Yaskawa INFORM job: 34.JBI

/JOB
//NAME 34
//POS
///NPOS 208,208,208,10,0,0
///TOOL 0
///POSTYPE PULSE
///PULSE
C00000=-36470,-76528,-106815,19279,71473,77234
C00001=-134470,-76528,-106815,19279,71473,77234
C00002=-159578,-94739,-111578,14965,102577,71346
C00003=-157881,-88069,-71686,3941,80760,68512
C00004=-158562,-88051,-67559,4028,78269,68198
C00005=-158841,-87937,-65852,4065,77294,68070
C00006=-158823,-87020,-63758,4076,76477,68050
C00007=-158841,-87937,-65852,4065,77294,68070
C00008=-158257,-85912,-63562,4020,76897,68259
C00009=-159408,-88670,-64664,4131,76218,67839
C00010=-158257,-85912,-63562,4020,76897,68259
C00011=-157986,-86044,-65280,3983,77870,68384
C00012=-157322,-86111,-69434,3896,80354,68691
C00013=-157948,-93050,-93119,3918,91369,68820
C00014=-158631,-94954,-89856,3971,88424,68498
C00015=-158911,-95544,-88477,3995,87288,68367
C00016=-158893,-95136,-86651,3995,86375,68344
C00017=-158911,-95544,-88477,3995,87288,68367
C00018=-158162,-93185,-86154,3931,87034,68613
C00019=-159307,-96640,-87495,4031,86143,68197
C00020=-158162,-93185,-86154,3931,87034,68613
C00021=-157891,-92621,-87539,3907,88161,68739
C00022=-157230,-90799,-90820,3855,91078,69051
C00023=-157971,-89638,-106553,4024,101368,69130
C00024=-158653,-94046,-104272,4030,97741,68787
C00025=-158932,-95549,-103251,4038,96357,68649
C00026=-158915,-95836,-101701,4026,95258,68619
C00027=-158932,-95549,-103251,4038,96357,68649
C00028=-158118,-93796,-101169,3964,95939,68906
C00029=-159263,-97999,-102797,4052,94839,68490
C00030=-158118,-93796,-101169,3964,95939,68906
C00031=-157847,-92365,-102209,3955,97297,69039
C00032=-157186,-88172,-104546,3946,100851,69371
C00033=-156260,-82084,-105550,20461,72444,69801
C00034=-137260,-84248,-120477,10166,77039,76482
C00035=11401,-148032,-125425,11667,16324,75771
C00036=126225,-114648,-117375,36487,17100,65054
C00037=168603,-127327,-105850,12339,78437,77405
C00038=188556,-88570,-70376,9474,73843,-79671
C00039=189658,-87934,-65982,9402,71368,-79472
C00040=190106,-87582,-64173,9375,70395,-79388
C00041=190093,-86631,-62058,9423,69594,-79456
C00042=190106,-87582,-64173,9375,70395,-79388
C00043=189092,-85833,-61994,9573,70077,-79779
C00044=190880,-87833,-62791,9297,69339,-79192
C00045=189092,-85833,-61994,9573,70077,-79779
C00046=188652,-86197,-63814,9595,71050,-79858
C00047=187573,-86869,-68234,9657,73522,-80046
C00048=174405,-91869,-88866,8360,85065,-80378
C00049=162023,-93599,-92534,7262,87848,-81242
C00050=162738,-95362,-89212,7186,84857,-81172
C00051=163031,-95900,-87810,7159,83700,-81138
C00052=163022,-95451,-85967,7171,82804,-81192
C00053=163031,-95900,-87810,7159,83700,-81138
C00054=162558,-93657,-85516,7221,83485,-81312
C00055=163728,-97065,-86834,7086,82448,-80971
C00056=162558,-93657,-85516,7221,83485,-81312
C00057=162272,-93147,-86925,7246,84631,-81343
C00058=161575,-91472,-90271,7318,87591,-81408
C00059=161833,-89597,-103823,7401,96799,-80781
C00060=162061,-91169,-106298,7358,97489,-80667
C00061=162777,-95345,-103917,7205,93844,-80645
C00062=163070,-96760,-102859,7152,92451,-80627
C00063=163061,-96969,-101279,7144,91380,-80691
C00064=163070,-96760,-102859,7152,92451,-80627
C00065=162549,-94558,-100616,7215,92250,-80812
C00066=163719,-98703,-102215,7058,91010,-80493
C00067=162549,-94558,-100616,7215,92250,-80812
C00068=162264,-93207,-101689,7266,93618,-80828
C00069=161567,-89224,-104115,7414,97191,-80847
C00070=161715,-86803,-103327,4886,98608,-77730
C00071=162141,-92472,-85533,-3463,86932,-68770
C00072=162126,-88781,-71814,-3762,80467,-68306
C00073=162843,-88708,-67661,-3852,77988,-67984
C00074=163137,-88572,-65944,-3890,77018,-67852
C00075=163128,-87638,-63844,-3901,76206,-67830
C00076=163137,-88572,-65944,-3890,77018,-67852
C00077=162593,-86370,-63634,-3847,76702,-68030
C00078=163767,-89113,-64727,-3960,76023,-67603
C00079=162593,-86370,-63634,-3847,76702,-68030
C00080=162306,-86518,-65359,-3809,77672,-68159
C00081=161607,-86627,-69532,-3720,80146,-68475
C00082=161949,-92223,-96357,-3744,93768,-68761
C00083=162073,-93836,-93212,-3726,91015,-68637
C00084=162789,-95666,-89915,-3783,88086,-68309
C00085=163083,-96227,-88523,-3809,86956,-68176
C00086=163074,-95793,-86687,-3810,86051,-68151
C00087=163083,-96227,-88523,-3809,86956,-68176
C00088=162687,-94151,-86288,-3775,86630,-68300
C00089=163864,-97585,-87612,-3878,85738,-67874
C00090=162687,-94151,-86288,-3775,86630,-68300
C00091=162400,-93622,-87691,-3749,87749,-68430
C00092=161699,-91892,-91016,-3692,90646,-68752
C00093=162002,-88104,-107646,-3859,102814,-69021
C00094=162113,-90810,-106745,-3822,100878,-68922
C00095=162829,-95111,-104412,-3836,97273,-68574
C00096=163122,-96572,-103371,-3847,95899,-68434
C00097=163114,-96817,-101805,-3837,94811,-68403
C00098=163122,-96572,-103371,-3847,95899,-68434
C00099=162678,-95201,-101447,-3805,95399,-68566
C00100=163858,-99394,-103055,-3897,94292,-68140
C00101=162678,-95201,-101447,-3805,95399,-68566
C00102=162391,-93819,-102511,-3793,96748,-68703
C00103=161689,-89747,-104911,-3775,100278,-69043
C00104=160138,-149166,-122708,-13309,73561,-68802
C00105=149595,-96211,-103761,-5489,101844,-74102
C00106=149594,-96505,-102316,-5465,100808,-74056
C00107=149006,-93113,-100988,-5479,101691,-74295
C00108=149599,-96300,-103483,-5484,101628,-74092
C00109=149598,-96527,-102324,-5465,100802,-74055
C00110=149603,-96557,-102335,-5465,100793,-74053
C00111=149607,-96579,-102343,-5465,100787,-74051
C00112=149608,-96287,-103789,-5489,101823,-74097
C00113=160720,-151449,-123129,-13814,72249,-68439
C00114=174899,-138237,-126795,1008,88740,-67536
C00115=163022,-96341,-102515,22398,105363,-76518
C00116=163017,-96713,-99258,22147,103326,-76913
C00117=163015,-96754,-97914,22060,102538,-77063
C00118=163022,-96736,-99152,22139,103253,-76925
C00119=162158,-93804,-96763,22109,103515,-77196
C00120=163010,-96735,-97907,22060,102545,-77064
C00121=163002,-96709,-97898,22061,102553,-77065
C00122=162997,-96690,-97891,22061,102560,-77066
C00123=162999,-96647,-99234,22149,103348,-76916
C00124=163003,-96272,-102489,22400,105387,-76520
C00125=163026,-93642,-108610,23163,110115,-75549
C00126=163006,-95534,-87485,21597,97146,-78065
C00127=163001,-94597,-83697,21497,95421,-78378
C00128=162999,-94160,-82153,21464,94744,-78500
C00129=163006,-94576,-83573,21494,95359,-78388
C00130=162142,-91714,-81191,21448,95589,-78662
C00131=162994,-94144,-82148,21463,94750,-78501
C00132=162986,-94123,-82140,21463,94758,-78503
C00133=162981,-94108,-82134,21463,94763,-78504
C00134=162983,-94543,-83678,21497,95441,-78382
C00135=162987,-95478,-87465,21598,97166,-78068
C00136=173072,-122981,-101575,-4997,88706,-65554
C00137=163055,-95539,-86908,782,102933,-69098
C00138=163053,-95162,-85345,779,102165,-69104
C00139=162194,-92631,-84353,657,102863,-69400
C00140=163060,-95514,-86735,782,102839,-69097
C00141=163059,-95178,-85351,779,102160,-69102
C00142=163066,-95200,-85359,780,102154,-69099
C00143=163072,-95216,-85365,781,102149,-69097
C00144=163073,-95594,-86928,784,102917,-69092
C00145=178442,-133591,-104623,-8068,82135,-63325
C00146=176542,-133362,-109369,-6755,86992,-64211
C00147=163036,-88875,-67291,2288,96831,-69180
C00148=163033,-87023,-63014,2278,95152,-69212
C00149=163032,-86242,-61276,2275,94484,-69224
C00150=162173,-84225,-60457,2128,95039,-69506
C00151=163038,-86971,-62872,2279,95091,-69211
C00152=163037,-86254,-61278,2276,94479,-69222
C00153=163044,-86268,-61280,2277,94473,-69220
C00154=163039,-85938,-60578,-1998,96244,-70315
C00155=163039,-86718,-62302,-2001,96904,-70326
C00156=163041,-88572,-66545,-2011,98562,-70352
C00157=163041,-94022,-81579,12660,98605,-75478
C00158=162985,-87715,-64806,21312,87868,-79725
C00159=162980,-85781,-60474,21324,86307,-80003
C00160=162979,-84969,-58714,21334,85685,-80113
C00161=162985,-85725,-60330,21325,86250,-80011
C00162=162122,-82990,-57905,21265,86391,-80297
C00163=162973,-84956,-58710,21333,85690,-80114
C00164=162965,-84939,-58703,21332,85696,-80116
C00165=162960,-84927,-58699,21332,85701,-80117
C00166=162962,-85738,-60458,21322,86323,-80007
C00167=162966,-87670,-64790,21310,87885,-79729
C00168=168603,-127327,-105850,12339,78437,77405
C00169=126225,-114648,-117375,36487,17100,65054
C00170=11401,-148032,-125425,11667,16324,75771
C00171=-137260,-84248,-120477,10166,77039,76482
C00172=-156260,-82084,-105550,20461,72444,69801
C00173=-171634,-136713,-119987,14813,82155,64373
C00174=-158729,-95167,-103646,5818,103191,69841
C00175=-158729,-95507,-102217,5790,102143,69791
C00176=-158743,-95268,-103371,5812,102972,69826
C00177=-157888,-92366,-100981,5813,102933,70115
C00178=-158724,-95485,-102217,5790,102154,69793
C00179=-158716,-95455,-102218,5791,102168,69796
C00180=-158711,-95433,-102218,5791,102179,69799
C00181=-158710,-95090,-103645,5820,103229,69849
C00182=-176787,-149067,-122219,18835,75411,61621
C00183=-173763,-146173,-128899,15065,83149,63746
C00184=-179123,-141279,-106647,10683,78126,61378
C00185=-158741,-94804,-86638,-974,104038,69307
C00186=-158742,-94449,-85096,-971,103271,69313
C00187=-158755,-94787,-86481,-976,103949,69303
C00188=-157900,-91912,-84097,-841,103969,69603
C00189=-158737,-94435,-85099,-970,103281,69315
C00190=-158729,-94416,-85104,-969,103293,69317
C00191=-158724,-94402,-85107,-968,103302,69319
C00192=-158723,-94755,-86649,-971,104070,69313
C00193=-179319,-141585,-106738,10818,77944,61288
C00194=-179127,-150966,-119474,10597,80994,61624
C00195=-158768,-88195,-66653,2364,98843,70558
C00196=-158769,-86372,-62416,2351,97173,70526
C00197=-158769,-85604,-60695,2347,96509,70514
C00198=-158782,-86330,-62292,2348,97119,70521
C00199=-157926,-83586,-59872,2521,97014,70811
C00200=-158763,-85596,-60701,2348,96517,70516
C00201=-158756,-85585,-60709,2349,96527,70518
C00202=-158750,-85577,-60715,2351,96535,70521
C00203=-158750,-86345,-62435,2355,97199,70533
C00204=-158749,-88164,-66671,2368,98869,70565
C00205=-159578,-94739,-111578,14965,102577,71346
C00206=-134470,-76528,-106815,19279,71473,77234
C00207=-36470,-76528,-106815,19279,71473,77234
BC00000=295325,674563,1075175
BC00001=353535,895977,1075175
BC00002=353535,975867,1075175
BC00003=382929,976652,1075175
BC00004=382929,976652,1075175
BC00005=382929,976652,1075175
BC00006=382929,976652,1075175
BC00007=382929,976652,1075175
BC00008=382929,976652,1075175
BC00009=382929,976652,1075175
BC00010=382929,976652,1075175
BC00011=382929,976652,1075175
BC00012=382929,976652,1075175
BC00013=382158,1006074,1075175
BC00014=382158,1006074,1075175
BC00015=382158,1006074,1075175
BC00016=382158,1006074,1075175
BC00017=382158,1006074,1075175
BC00018=382158,1006074,1075175
BC00019=382158,1006074,1075175
BC00020=382158,1006074,1075175
BC00021=382158,1006074,1075175
BC00022=382158,1006074,1075175
BC00023=381896,1032866,1075175
BC00024=381896,1032866,1075175
BC00025=381896,1032866,1075175
BC00026=381896,1032866,1075175
BC00027=381896,1032866,1075175
BC00028=381896,1032866,1075175
BC00029=381896,1032866,1075175
BC00030=381896,1032866,1075175
BC00031=381896,1032866,1075175
BC00032=381896,1032866,1075175
BC00033=381896,966588,1075175
BC00034=353816,923989,1075175
BC00035=398190,1030285,1075175
BC00036=312632,1138057,1075175
BC00037=340753,1115300,1075175
BC00038=340753,1115300,1075175
BC00039=340753,1115300,1075175
BC00040=340753,1115300,1075175
BC00041=340753,1115300,1075175
BC00042=340753,1115300,1075175
BC00043=340753,1115300,1075175
BC00044=340753,1115300,1075175
BC00045=340753,1115300,1075175
BC00046=340753,1115300,1075175
BC00047=340753,1115300,1075175
BC00048=322796,1114285,1075175
BC00049=305962,1113333,1075175
BC00050=305962,1113333,1075175
BC00051=305962,1113333,1075175
BC00052=305962,1113333,1075175
BC00053=305962,1113333,1075175
BC00054=305962,1113333,1075175
BC00055=305962,1113333,1075175
BC00056=305962,1113333,1075175
BC00057=305962,1113333,1075175
BC00058=305962,1113333,1075175
BC00059=305642,1099956,1075175
BC00060=305321,1086579,1075175
BC00061=305321,1086579,1075175
BC00062=305321,1086579,1075175
BC00063=305321,1086579,1075175
BC00064=305321,1086579,1075175
BC00065=305321,1086579,1075175
BC00066=305321,1086579,1075175
BC00067=305321,1086579,1075175
BC00068=305321,1086579,1075175
BC00069=305321,1086579,1075175
BC00070=323405,1100688,1075175
BC00071=381464,1145987,1075175
BC00072=383367,1147472,1075175
BC00073=383367,1147472,1075175
BC00074=383367,1147472,1075175
BC00075=383367,1147472,1075175
BC00076=383367,1147472,1075175
BC00077=383367,1147472,1075175
BC00078=383367,1147472,1075175
BC00079=383367,1147472,1075175
BC00080=383367,1147472,1075175
BC00081=383367,1147472,1075175
BC00082=383362,1127243,1075175
BC00083=383359,1117611,1075175
BC00084=383359,1117611,1075175
BC00085=383359,1117611,1075175
BC00086=383359,1117611,1075175
BC00087=383359,1117611,1075175
BC00088=383359,1117611,1075175
BC00089=383359,1117611,1075175
BC00090=383359,1117611,1075175
BC00091=383359,1117611,1075175
BC00092=383359,1117611,1075175
BC00093=383208,1098974,1075175
BC00094=383141,1090691,1075175
BC00095=383141,1090691,1075175
BC00096=383141,1090691,1075175
BC00097=383141,1090691,1075175
BC00098=383141,1090691,1075175
BC00099=383141,1090691,1075175
BC00100=383141,1090691,1075175
BC00101=383141,1090691,1075175
BC00102=383141,1090691,1075175
BC00103=383141,1090691,1075175
BC00104=347951,1086630,1075175
BC00105=348637,1089204,1075175
BC00106=348912,1090234,1075175
BC00107=348912,1090234,1075175
BC00108=348912,1090234,1075175
BC00109=353690,1090245,1075175
BC00110=360061,1090261,1075175
BC00111=364840,1090272,1075175
BC00112=364565,1089242,1075175
BC00113=363879,1086668,1075175
BC00114=346096,1068466,1075175
BC00115=323525,1045363,1075175
BC00116=322819,1049711,1075175
BC00117=322536,1051450,1075175
BC00118=322536,1051450,1075175
BC00119=322536,1051450,1075175
BC00120=317758,1051439,1075175
BC00121=311387,1051424,1075175
BC00122=306609,1051412,1075175
BC00123=306891,1049673,1075175
BC00124=307598,1045324,1075175
BC00125=309359,1048307,1075175
BC00126=323451,1072164,1075175
BC00127=322745,1076512,1075175
BC00128=322462,1078251,1075175
BC00129=322462,1078251,1075175
BC00130=322462,1078251,1075175
BC00131=317684,1078240,1075175
BC00132=311313,1078225,1075175
BC00133=306534,1078213,1075175
BC00134=306817,1076474,1075175
BC00135=307523,1072125,1075175
BC00136=364639,1081055,1075175
BC00137=365322,1085072,1075175
BC00138=365595,1086678,1075175
BC00139=365595,1086678,1075175
BC00140=365595,1086678,1075175
BC00141=370373,1086690,1075175
BC00142=376744,1086705,1075175
BC00143=381523,1086717,1075175
BC00144=381250,1085110,1075175
BC00145=380567,1081094,1075175
BC00146=378567,1084057,1075175
BC00147=364571,1104797,1075175
BC00148=365253,1109149,1075175
BC00149=365525,1110890,1075175
BC00150=365525,1110890,1075175
BC00151=365525,1110890,1075175
BC00152=370304,1110904,1075175
BC00153=376537,1110923,1075175
BC00154=371992,1111607,1075175
BC00155=371443,1109885,1075175
BC00156=370073,1105582,1075175
BC00157=341083,1103324,1075175
BC00158=323368,1101944,1075175
BC00159=322661,1106292,1075175
BC00160=322379,1108032,1075175
BC00161=322379,1108032,1075175
BC00162=322379,1108032,1075175
BC00163=317600,1108020,1075175
BC00164=311229,1108005,1075175
BC00165=306451,1107994,1075175
BC00166=306733,1106254,1075175
BC00167=307440,1101906,1075175
BC00168=340753,1115300,1075175
BC00169=312632,1138057,1075175
BC00170=398190,1030285,1075175
BC00171=353816,923989,1075175
BC00172=381896,966588,1075175
BC00173=363636,1044565,1075175
BC00174=364364,1042023,1075175
BC00175=364655,1041006,1075175
BC00176=364655,1041006,1075175
BC00177=364655,1041006,1075175
BC00178=369433,1041019,1075175
BC00179=375804,1041036,1075175
BC00180=380582,1041048,1075175
BC00181=380291,1042065,1075175
BC00182=379563,1044606,1075175
BC00183=363636,1044565,1075175
BC00184=363753,1044796,1075175
BC00185=364482,1040696,1075175
BC00186=364774,1039056,1075175
BC00187=364774,1039056,1075175
BC00188=364774,1039056,1075175
BC00189=369552,1039069,1075175
BC00190=375923,1039086,1075175
BC00191=380702,1039098,1075175
BC00192=380410,1040738,1075175
BC00193=379681,1044838,1075175
BC00194=363753,1044796,1075175
BC00195=353535,1018425,1075175
BC00196=354953,1014154,1075175
BC00197=355520,1012445,1075175
BC00198=355520,1012445,1075175
BC00199=355520,1012445,1075175
BC00200=360298,1012458,1075175
BC00201=366669,1012474,1075175
BC00202=371447,1012487,1075175
BC00203=370880,1014195,1075175
BC00204=369462,1018467,1075175
BC00205=353535,975867,1075175
BC00206=353535,895977,1075175
BC00207=295325,674563,1075175
EC00000=-1418945,-556475
EC00001=-1418945,-556475
EC00002=-1418945,-556475
EC00003=-1418945,-556475
EC00004=-1418945,-556475
EC00005=-1418945,-556475
EC00006=-1418945,-556475
EC00007=-1418945,-556475
EC00008=-1418945,-556475
EC00009=-1418945,-556475
EC00010=-1418945,-556475
EC00011=-1418945,-556475
EC00012=-1418945,-556475
EC00013=-1418945,-556475
EC00014=-1418945,-556475
EC00015=-1418945,-556475
EC00016=-1418945,-556475
EC00017=-1418945,-556475
EC00018=-1418945,-556475
EC00019=-1418945,-556475
EC00020=-1418945,-556475
EC00021=-1418945,-556475
EC00022=-1418945,-556475
EC00023=-1418945,-556475
EC00024=-1418945,-556475
EC00025=-1418945,-556475
EC00026=-1418945,-556475
EC00027=-1418945,-556475
EC00028=-1418945,-556475
EC00029=-1418945,-556475
EC00030=-1418945,-556475
EC00031=-1418945,-556475
EC00032=-1418945,-556475
EC00033=-1418945,-556475
EC00034=-1418945,-556475
EC00035=-1595090,-3837
EC00036=-1773681,556475
EC00037=-1773681,556475
EC00038=-1773681,556475
EC00039=-1773681,556475
EC00040=-1773681,556475
EC00041=-1773681,556475
EC00042=-1773681,556475
EC00043=-1773681,556475
EC00044=-1773681,556475
EC00045=-1773681,556475
EC00046=-1773681,556475
EC00047=-1773681,556475
EC00048=-1773681,556475
EC00049=-1773681,556475
EC00050=-1773681,556475
EC00051=-1773681,556475
EC00052=-1773681,556475
EC00053=-1773681,556475
EC00054=-1773681,556475
EC00055=-1773681,556475
EC00056=-1773681,556475
EC00057=-1773681,556475
EC00058=-1773681,556475
EC00059=-1773681,556475
EC00060=-1773681,556475
EC00061=-1773681,556475
EC00062=-1773681,556475
EC00063=-1773681,556475
EC00064=-1773681,556475
EC00065=-1773681,556475
EC00066=-1773681,556475
EC00067=-1773681,556475
EC00068=-1773681,556475
EC00069=-1773681,556475
EC00070=-1773681,556475
EC00071=-1773681,556475
EC00072=-1773681,556475
EC00073=-1773681,556475
EC00074=-1773681,556475
EC00075=-1773681,556475
EC00076=-1773681,556475
EC00077=-1773681,556475
EC00078=-1773681,556475
EC00079=-1773681,556475
EC00080=-1773681,556475
EC00081=-1773681,556475
EC00082=-1773681,556475
EC00083=-1773681,556475
EC00084=-1773681,556475
EC00085=-1773681,556475
EC00086=-1773681,556475
EC00087=-1773681,556475
EC00088=-1773681,556475
EC00089=-1773681,556475
EC00090=-1773681,556475
EC00091=-1773681,556475
EC00092=-1773681,556475
EC00093=-1773681,556475
EC00094=-1773681,556475
EC00095=-1773681,556475
EC00096=-1773681,556475
EC00097=-1773681,556475
EC00098=-1773681,556475
EC00099=-1773681,556475
EC00100=-1773681,556475
EC00101=-1773681,556475
EC00102=-1773681,556475
EC00103=-1773681,556475
EC00104=-1773681,556475
EC00105=-1773681,556475
EC00106=-1773681,556475
EC00107=-1773681,556475
EC00108=-1773681,556475
EC00109=-1773681,556475
EC00110=-1773681,556475
EC00111=-1773681,556475
EC00112=-1773681,556475
EC00113=-1773681,556475
EC00114=-1773681,556475
EC00115=-1773681,556475
EC00116=-1773681,556475
EC00117=-1773681,556475
EC00118=-1773681,556475
EC00119=-1773681,556475
EC00120=-1773681,556475
EC00121=-1773681,556475
EC00122=-1773681,556475
EC00123=-1773681,556475
EC00124=-1773681,556475
EC00125=-1773681,556475
EC00126=-1773681,556475
EC00127=-1773681,556475
EC00128=-1773681,556475
EC00129=-1773681,556475
EC00130=-1773681,556475
EC00131=-1773681,556475
EC00132=-1773681,556475
EC00133=-1773681,556475
EC00134=-1773681,556475
EC00135=-1773681,556475
EC00136=-1773681,556475
EC00137=-1773681,556475
EC00138=-1773681,556475
EC00139=-1773681,556475
EC00140=-1773681,556475
EC00141=-1773681,556475
EC00142=-1773681,556475
EC00143=-1773681,556475
EC00144=-1773681,556475
EC00145=-1773681,556475
EC00146=-1773681,556475
EC00147=-1773681,556475
EC00148=-1773681,556475
EC00149=-1773681,556475
EC00150=-1773681,556475
EC00151=-1773681,556475
EC00152=-1773681,556475
EC00153=-1773681,556475
EC00154=-1773681,556475
EC00155=-1773681,556475
EC00156=-1773681,556475
EC00157=-1773681,556475
EC00158=-1773681,556475
EC00159=-1773681,556475
EC00160=-1773681,556475
EC00161=-1773681,556475
EC00162=-1773681,556475
EC00163=-1773681,556475
EC00164=-1773681,556475
EC00165=-1773681,556475
EC00166=-1773681,556475
EC00167=-1773681,556475
EC00168=-1773681,556475
EC00169=-1773681,556475
EC00170=-1595090,-3837
EC00171=-1418945,-556475
EC00172=-1418945,-556475
EC00173=-1418945,-556475
EC00174=-1418945,-556475
EC00175=-1418945,-556475
EC00176=-1418945,-556475
EC00177=-1418945,-556475
EC00178=-1418945,-556475
EC00179=-1418945,-556475
EC00180=-1418945,-556475
EC00181=-1418945,-556475
EC00182=-1418945,-556475
EC00183=-1418945,-556475
EC00184=-1418945,-556475
EC00185=-1418945,-556475
EC00186=-1418945,-556475
EC00187=-1418945,-556475
EC00188=-1418945,-556475
EC00189=-1418945,-556475
EC00190=-1418945,-556475
EC00191=-1418945,-556475
EC00192=-1418945,-556475
EC00193=-1418945,-556475
EC00194=-1418945,-556475
EC00195=-1418945,-556475
EC00196=-1418945,-556475
EC00197=-1418945,-556475
EC00198=-1418945,-556475
EC00199=-1418945,-556475
EC00200=-1418945,-556475
EC00201=-1418945,-556475
EC00202=-1418945,-556475
EC00203=-1418945,-556475
EC00204=-1418945,-556475
EC00205=-1418945,-556475
EC00206=-1418945,-556475
EC00207=-1418945,-556475
///POSTYPE BASE
///RECTAN
///RCONF 0,0,0,0,0,0,0,0,0,0,0,0,0,0,0,0,0,0,0,0,0,0,0,0
P00006=-0.339,1.359,3.368,0.0000,0.0000,0.0000
P00021=-0.339,1.359,3.368,0.0000,0.0000,0.0000
P00022=-0.114,-0.780,3.887,0.0000,0.0000,0.0000
P00023=0.297,-0.076,-2.402,0.0000,0.0000,0.0000
P00031=1.853,-0.001,-1.549,0.0000,0.0000,0.0000
P00032=1.957,0.503,-7.217,0.0000,0.0000,0.0000
///RCONF 0,0,0,0,1,0,0,0,0,0,0,0,0,0,0,0,0,0,0,0,0,0,0,0
P00033=-0.123,0.612,-5.012,0.0000,0.0000,0.0000
///RCONF 0,0,0,0,0,0,0,0,0,0,0,0,0,0,0,0,0,0,0,0,0,0,0,0
P00034=-0.304,0.773,-2.693,0.0000,0.0000,0.0000
P00035=2.817,0.591,-1.622,0.0000,0.0000,0.0000
P00036=-1.108,-0.829,1.850,0.0000,0.0000,0.0000
//INST
///DATE 2024/01/19 10:04
///ATTR SC,RW
///GROUP1 RB1,BS1
///GROUP2 ST1
NOP
'OK_r2_O7.1(P)(-160.-90)new
MOVJ C00000 BC00000 VJ=100.00  +MOVJ EC00000 VJ=100.00
MOVJ C00001 BC00001 VJ=100.00  +MOVJ EC00001 VJ=100.00
MOVJ C00002 BC00002 VJ=100.00  +MOVJ EC00002 VJ=100.00
'Path S1422
SSFTOF
MOVJ C00003 BC00003 VJ=100.00  +MOVJ EC00003 VJ=100.00
MOVL C00004 BC00004 V=400.0  +MOVJ EC00004 VJ=100.00
SMOVL C00005 BC00005 V=60.0  +MOVJ EC00005
SREFP 3 C00006 BC00006  +REFP EC00006
CALL JOB:SEARCH-R1-S1
SET P021 P006
SSFTON P021
SMOVL C00007 BC00007 V=60.0  +MOVJ EC00007
SMOVL C00008 BC00008 V=60.0  +MOVJ EC00008
SREFP 3 C00009 BC00009  +REFP EC00009
CALL JOB:SEARCH-R1-S1
SET P021 P006
SSFTON P021
SMOVL C00010 BC00010 V=60.0  +MOVJ EC00010
MOVL C00011 BC00011 V=400.0  +MOVJ EC00011 VJ=100.00
MOVL C00012 BC00012 V=1000.0  +MOVJ EC00012 VJ=100.00
'Path S1423
SSFTOF
MOVJ C00013 BC00013 VJ=100.00  +MOVJ EC00013 VJ=100.00
MOVL C00014 BC00014 V=400.0  +MOVJ EC00014 VJ=100.00
SMOVL C00015 BC00015 V=60.0  +MOVJ EC00015
SREFP 3 C00016 BC00016  +REFP EC00016
CALL JOB:SEARCH-R1-S1
SET P022 P006
SSFTON P022
SMOVL C00017 BC00017 V=60.0  +MOVJ EC00017
SMOVL C00018 BC00018 V=60.0  +MOVJ EC00018
SREFP 3 C00019 BC00019  +REFP EC00019
CALL JOB:SEARCH-R1-S1
SET P022 P006
SSFTON P022
SMOVL C00020 BC00020 V=60.0  +MOVJ EC00020
MOVL C00021 BC00021 V=400.0  +MOVJ EC00021 VJ=100.00
MOVL C00022 BC00022 V=1000.0  +MOVJ EC00022 VJ=100.00
'Path S1424
SSFTOF
MOVJ C00023 BC00023 VJ=100.00  +MOVJ EC00023 VJ=100.00
MOVL C00024 BC00024 V=400.0  +MOVJ EC00024 VJ=100.00
SMOVL C00025 BC00025 V=60.0  +MOVJ EC00025
SREFP 3 C00026 BC00026  +REFP EC00026
CALL JOB:SEARCH-R1-S1
SET P023 P006
SSFTON P023
SMOVL C00027 BC00027 V=60.0  +MOVJ EC00027
SMOVL C00028 BC00028 V=60.0  +MOVJ EC00028
SREFP 3 C00029 BC00029  +REFP EC00029
CALL JOB:SEARCH-R1-S1
SET P023 P006
SSFTON P023
SMOVL C00030 BC00030 V=60.0  +MOVJ EC00030
MOVL C00031 BC00031 V=400.0  +MOVJ EC00031 VJ=100.00
MOVL C00032 BC00032 V=1000.0  +MOVJ EC00032 VJ=100.00
'obrot
MOVJ C00033 BC00033 VJ=100.00  +MOVJ EC00033 VJ=100.00
MOVJ C00034 BC00034 VJ=100.00  +MOVJ EC00034 VJ=100.00
MOVJ C00035 BC00035 VJ=100.00  +MOVJ EC00035 VJ=100.00
MOVJ C00036 BC00036 VJ=100.00  +MOVJ EC00036 VJ=100.00
MOVJ C00037 BC00037 VJ=100.00  +MOVJ EC00037 VJ=100.00
'Path S1077
SSFTOF
MOVJ C00038 BC00038 VJ=100.00  +MOVJ EC00038 VJ=100.00
MOVL C00039 BC00039 V=400.0  +MOVJ EC00039 VJ=100.00
SMOVL C00040 BC00040 V=60.0  +MOVJ EC00040
SREFP 3 C00041 BC00041  +REFP EC00041
CALL JOB:SEARCH-R1-S1
SET P031 P006
SSFTON P031
SMOVL C00042 BC00042 V=60.0  +MOVJ EC00042
SMOVL C00043 BC00043 V=60.0  +MOVJ EC00043
SREFP 3 C00044 BC00044  +REFP EC00044
CALL JOB:SEARCH-R1-S1
SET P031 P006
SSFTON P031
SMOVL C00045 BC00045 V=60.0  +MOVJ EC00045
MOVL C00046 BC00046 V=400.0  +MOVJ EC00046 VJ=100.00
MOVL C00047 BC00047 V=1000.0  +MOVJ EC00047 VJ=100.00
MOVJ C00048 BC00048 VJ=100.00  +MOVJ EC00048 VJ=100.00
'Path S1078
SSFTOF
MOVJ C00049 BC00049 VJ=100.00  +MOVJ EC00049 VJ=100.00
MOVL C00050 BC00050 V=400.0  +MOVJ EC00050 VJ=100.00
SMOVL C00051 BC00051 V=60.0  +MOVJ EC00051
SREFP 3 C00052 BC00052  +REFP EC00052
CALL JOB:SEARCH-R1-S1
SET P032 P006
SSFTON P032
SMOVL C00053 BC00053 V=60.0  +MOVJ EC00053
SMOVL C00054 BC00054 V=60.0  +MOVJ EC00054
SREFP 3 C00055 BC00055  +REFP EC00055
CALL JOB:SEARCH-R1-S1
SET P032 P006
SSFTON P032
SMOVL C00056 BC00056 V=60.0  +MOVJ EC00056
MOVL C00057 BC00057 V=400.0  +MOVJ EC00057 VJ=100.00
MOVL C00058 BC00058 V=1000.0  +MOVJ EC00058 VJ=100.00
MOVJ C00059 BC00059 VJ=100.00  +MOVJ EC00059 VJ=100.00
'Path S1079
SSFTOF
MOVJ C00060 BC00060 VJ=100.00  +MOVJ EC00060 VJ=100.00
MOVL C00061 BC00061 V=400.0  +MOVJ EC00061 VJ=100.00
SMOVL C00062 BC00062 V=60.0  +MOVJ EC00062
SREFP 3 C00063 BC00063  +REFP EC00063
CALL JOB:SEARCH-R1-S1
SET P033 P006
SSFTON P033
SMOVL C00064 BC00064 V=60.0  +MOVJ EC00064
SMOVL C00065 BC00065 V=60.0  +MOVJ EC00065
SREFP 3 C00066 BC00066  +REFP EC00066
CALL JOB:SEARCH-R1-S1
SET P033 P006
SSFTON P033
SMOVL C00067 BC00067 V=60.0  +MOVJ EC00067
MOVL C00068 BC00068 V=400.0  +MOVJ EC00068 VJ=100.00
MOVL C00069 BC00069 V=1000.0  +MOVJ EC00069 VJ=100.00
MOVJ C00070 BC00070 VJ=100.00  +MOVJ EC00070 VJ=100.00
MOVJ C00071 BC00071 VJ=100.00  +MOVJ EC00071 VJ=100.00
'Path S1080
SSFTOF
MOVJ C00072 BC00072 VJ=100.00  +MOVJ EC00072 VJ=100.00
MOVL C00073 BC00073 V=400.0  +MOVJ EC00073 VJ=100.00
SMOVL C00074 BC00074 V=60.0  +MOVJ EC00074
SREFP 3 C00075 BC00075  +REFP EC00075
CALL JOB:SEARCH-R1-S1
SET P034 P006
SSFTON P034
SMOVL C00076 BC00076 V=60.0  +MOVJ EC00076
SMOVL C00077 BC00077 V=60.0  +MOVJ EC00077
SREFP 3 C00078 BC00078  +REFP EC00078
CALL JOB:SEARCH-R1-S1
SET P034 P006
SSFTON P034
SMOVL C00079 BC00079 V=60.0  +MOVJ EC00079
MOVL C00080 BC00080 V=400.0  +MOVJ EC00080 VJ=100.00
MOVL C00081 BC00081 V=1000.0  +MOVJ EC00081 VJ=100.00
MOVJ C00082 BC00082 VJ=100.00  +MOVJ EC00082 VJ=100.00
'Path S1081
SSFTOF
MOVJ C00083 BC00083 VJ=100.00  +MOVJ EC00083 VJ=100.00
MOVL C00084 BC00084 V=400.0  +MOVJ EC00084 VJ=100.00
SMOVL C00085 BC00085 V=60.0  +MOVJ EC00085
SREFP 3 C00086 BC00086  +REFP EC00086
CALL JOB:SEARCH-R1-S1
SET P035 P006
SSFTON P035
SMOVL C00087 BC00087 V=60.0  +MOVJ EC00087
SMOVL C00088 BC00088 V=60.0  +MOVJ EC00088
SREFP 3 C00089 BC00089  +REFP EC00089
CALL JOB:SEARCH-R1-S1
SET P035 P006
SSFTON P035
SMOVL C00090 BC00090 V=60.0  +MOVJ EC00090
MOVL C00091 BC00091 V=400.0  +MOVJ EC00091 VJ=100.00
MOVL C00092 BC00092 V=1000.0  +MOVJ EC00092 VJ=100.00
MOVJ C00093 BC00093 VJ=100.00  +MOVJ EC00093 VJ=100.00
'Path S1082
SSFTOF
MOVJ C00094 BC00094 VJ=100.00  +MOVJ EC00094 VJ=100.00
MOVL C00095 BC00095 V=400.0  +MOVJ EC00095 VJ=100.00
SMOVL C00096 BC00096 V=60.0  +MOVJ EC00096
SREFP 3 C00097 BC00097  +REFP EC00097
CALL JOB:SEARCH-R1-S1
SET P036 P006
SSFTON P036
SMOVL C00098 BC00098 V=60.0  +MOVJ EC00098
SMOVL C00099 BC00099 V=60.0  +MOVJ EC00099
SREFP 3 C00100 BC00100  +REFP EC00100
CALL JOB:SEARCH-R1-S1
SET P036 P006
SSFTON P036
SMOVL C00101 BC00101 V=60.0  +MOVJ EC00101
MOVL C00102 BC00102 V=400.0  +MOVJ EC00102 VJ=100.00
MOVL C00103 BC00103 V=1000.0  +MOVJ EC00103 VJ=100.00
'Path W260
SSFTOF
SSFTON P036
MOVJ C00104 BC00104 VJ=100.00  +MOVJ EC00104 VJ=100.00
SMOVL C00105 BC00105 V=400.0  +MOVJ EC00105
SMOVL C00106 BC00106 V=100.0 PL=0  +MOVJ EC00106
SREFP 1 C00107 BC00107  +REFP EC00107
SREFP 2 C00108 BC00108  +REFP EC00108
MACRO1 MJ#(0) ARGF0
ARCON
SMOVL C00109 BC00109 V=10.0  +MOVJ EC00109
SMOVL C00110 BC00110 V=10.0  +MOVJ EC00110
SMOVL C00111 BC00111 V=10.0  +MOVJ EC00111
ARCOF
SMOVL C00112 BC00112 V=400.0  +MOVJ EC00112
SMOVL C00113 BC00113 V=1000.0  +MOVJ EC00113
SSFTOF
MOVJ C00114 BC00114 VJ=100.00  +MOVJ EC00114 VJ=100.00
'Path W261
SSFTOF
SSFTON P033
MOVJ C00115 BC00115 VJ=100.00  +MOVJ EC00115 VJ=100.00
SMOVL C00116 BC00116 V=400.0  +MOVJ EC00116
SMOVL C00117 BC00117 V=100.0 PL=0  +MOVJ EC00117
SREFP 1 C00118 BC00118  +REFP EC00118
SREFP 2 C00119 BC00119  +REFP EC00119
MACRO1 MJ#(0) ARGF0
ARCON
SMOVL C00120 BC00120 V=10.0  +MOVJ EC00120
SMOVL C00121 BC00121 V=10.0  +MOVJ EC00121
SMOVL C00122 BC00122 V=10.0  +MOVJ EC00122
ARCOF
SMOVL C00123 BC00123 V=400.0  +MOVJ EC00123
SMOVL C00124 BC00124 V=1000.0  +MOVJ EC00124
SSFTOF
MOVJ C00125 BC00125 VJ=100.00  +MOVJ EC00125 VJ=100.00
'Path W1083
SSFTOF
SSFTON P032
MOVJ C00126 BC00126 VJ=100.00  +MOVJ EC00126 VJ=100.00
SMOVL C00127 BC00127 V=400.0  +MOVJ EC00127
SMOVL C00128 BC00128 V=100.0 PL=0  +MOVJ EC00128
SREFP 1 C00129 BC00129  +REFP EC00129
SREFP 2 C00130 BC00130  +REFP EC00130
MACRO1 MJ#(0) ARGF0
ARCON
SMOVL C00131 BC00131 V=10.0  +MOVJ EC00131
SMOVL C00132 BC00132 V=10.0  +MOVJ EC00132
SMOVL C00133 BC00133 V=10.0  +MOVJ EC00133
ARCOF
SMOVL C00134 BC00134 V=400.0  +MOVJ EC00134
SMOVL C00135 BC00135 V=1000.0  +MOVJ EC00135
SSFTOF
'Path W262
SSFTOF
SSFTON P035
MOVJ C00136 BC00136 VJ=100.00  +MOVJ EC00136 VJ=100.00
SMOVL C00137 BC00137 V=400.0  +MOVJ EC00137
SMOVL C00138 BC00138 V=100.0 PL=0  +MOVJ EC00138
SREFP 1 C00139 BC00139  +REFP EC00139
SREFP 2 C00140 BC00140  +REFP EC00140
MACRO1 MJ#(0) ARGF0
ARCON
SMOVL C00141 BC00141 V=10.0  +MOVJ EC00141
SMOVL C00142 BC00142 V=10.0  +MOVJ EC00142
SMOVL C00143 BC00143 V=10.0  +MOVJ EC00143
ARCOF
SMOVL C00144 BC00144 V=400.0  +MOVJ EC00144
SMOVL C00145 BC00145 V=1000.0  +MOVJ EC00145
SSFTOF
MOVJ C00146 BC00146 VJ=100.00  +MOVJ EC00146 VJ=100.00
'Path W264
SSFTOF
SSFTON P034
MOVJ C00147 BC00147 VJ=100.00  +MOVJ EC00147 VJ=100.00
SMOVL C00148 BC00148 V=400.0  +MOVJ EC00148
SMOVL C00149 BC00149 V=100.0 PL=0  +MOVJ EC00149
SREFP 1 C00150 BC00150  +REFP EC00150
SREFP 2 C00151 BC00151  +REFP EC00151
MACRO1 MJ#(0) ARGF0
ARCON
SMOVL C00152 BC00152 V=10.0  +MOVJ EC00152
SMOVL C00153 BC00153 V=10.0  +MOVJ EC00153
SMOVL C00154 BC00154 V=10.0  +MOVJ EC00154
ARCOF
SMOVL C00155 BC00155 V=400.0  +MOVJ EC00155
SMOVL C00156 BC00156 V=1000.0  +MOVJ EC00156
SSFTOF
MOVJ C00157 BC00157 VJ=100.00  +MOVJ EC00157 VJ=100.00
'Path W263
SSFTOF
SSFTON P031
MOVJ C00158 BC00158 VJ=100.00  +MOVJ EC00158 VJ=100.00
SMOVL C00159 BC00159 V=400.0  +MOVJ EC00159
SMOVL C00160 BC00160 V=100.0 PL=0  +MOVJ EC00160
SREFP 1 C00161 BC00161  +REFP EC00161
SREFP 2 C00162 BC00162  +REFP EC00162
MACRO1 MJ#(0) ARGF0
ARCON
SMOVL C00163 BC00163 V=10.0  +MOVJ EC00163
SMOVL C00164 BC00164 V=10.0  +MOVJ EC00164
SMOVL C00165 BC00165 V=10.0  +MOVJ EC00165
ARCOF
SMOVL C00166 BC00166 V=400.0  +MOVJ EC00166
SMOVL C00167 BC00167 V=1000.0  +MOVJ EC00167
SSFTOF
'obrot
MOVJ C00168 BC00168 VJ=100.00  +MOVJ EC00168 VJ=100.00
MOVJ C00169 BC00169 VJ=100.00  +MOVJ EC00169 VJ=100.00
MOVJ C00170 BC00170 VJ=100.00  +MOVJ EC00170 VJ=100.00
MOVJ C00171 BC00171 VJ=100.00  +MOVJ EC00171 VJ=100.00
MOVJ C00172 BC00172 VJ=100.00  +MOVJ EC00172 VJ=100.00
'Path W1425
SSFTOF
SSFTON P023
MOVJ C00173 BC00173 VJ=100.00  +MOVJ EC00173 VJ=100.00
SMOVL C00174 BC00174 V=100.0  +MOVJ EC00174
SMOVL C00175 BC00175 V=100.0 PL=0  +MOVJ EC00175
SREFP 1 C00176 BC00176  +REFP EC00176
SREFP 2 C00177 BC00177  +REFP EC00177
MACRO1 MJ#(0) ARGF0
ARCON
SMOVL C00178 BC00178 V=10.0  +MOVJ EC00178
SMOVL C00179 BC00179 V=10.0  +MOVJ EC00179
SMOVL C00180 BC00180 V=10.0  +MOVJ EC00180
ARCOF
SMOVL C00181 BC00181 V=400.0  +MOVJ EC00181
SMOVL C00182 BC00182 V=1000.0  +MOVJ EC00182
SSFTOF
MOVJ C00183 BC00183 VJ=100.00  +MOVJ EC00183 VJ=100.00
'Path W1426
SSFTOF
SSFTON P022
MOVJ C00184 BC00184 VJ=100.00  +MOVJ EC00184 VJ=100.00
SMOVL C00185 BC00185 V=100.0  +MOVJ EC00185
SMOVL C00186 BC00186 V=100.0 PL=0  +MOVJ EC00186
SREFP 1 C00187 BC00187  +REFP EC00187
SREFP 2 C00188 BC00188  +REFP EC00188
MACRO1 MJ#(0) ARGF0
ARCON
SMOVL C00189 BC00189 V=10.0  +MOVJ EC00189
SMOVL C00190 BC00190 V=10.0  +MOVJ EC00190
SMOVL C00191 BC00191 V=10.0  +MOVJ EC00191
ARCOF
SMOVL C00192 BC00192 V=400.0  +MOVJ EC00192
SMOVL C00193 BC00193 V=1000.0  +MOVJ EC00193
SSFTOF
MOVJ C00194 BC00194 VJ=100.00  +MOVJ EC00194 VJ=100.00
'Path W1427
SSFTOF
SSFTON P021
MOVJ C00195 BC00195 VJ=100.00  +MOVJ EC00195 VJ=100.00
SMOVL C00196 BC00196 V=100.0  +MOVJ EC00196
SMOVL C00197 BC00197 V=100.0 PL=0  +MOVJ EC00197
SREFP 1 C00198 BC00198  +REFP EC00198
SREFP 2 C00199 BC00199  +REFP EC00199
MACRO1 MJ#(0) ARGF0
ARCON
SMOVL C00200 BC00200 V=10.0  +MOVJ EC00200
SMOVL C00201 BC00201 V=10.0  +MOVJ EC00201
SMOVL C00202 BC00202 V=10.0  +MOVJ EC00202
ARCOF
SMOVL C00203 BC00203 V=400.0  +MOVJ EC00203
SMOVL C00204 BC00204 V=1000.0  +MOVJ EC00204
SSFTOF
MOVJ C00205 BC00205 VJ=100.00  +MOVJ EC00205 VJ=100.00
MOVJ C00206 BC00206 VJ=100.00  +MOVJ EC00206 VJ=100.00
MOVJ C00207 BC00207 VJ=100.00  +MOVJ EC00207 VJ=100.00
END
